PROGRAM MAIN
VAR
	concrete				:ConcreteAssertions();
	tests					:CNM_AssertionInterfaceTests.AssertionTester(concrete);
END_VAR

TcUnit.RUN_IN_SEQUENCE();

END_PROGRAM

(* stored: Version 1.1.0.1, ProductVersion 3.1.4024.12
   POU MAIN: Id {88f0f169-9aec-448c-9545-39ea6c60d390}, SpecialFunc None *)
